PROGRAM ST_ComponentDescriptor
VAR
END_VAR

END_PROGRAM

(* stored: Version 1.1.0.1
   POU ST_ComponentDescriptor: Id {91c36fa3-bacd-42e1-9ae3-cc8732ed5933}, SpecialFunc None *)
